FUNCTION_BLOCK FB_HeatPump EXTENDS FB_Actor2Point
VAR_INPUT
END_VAR
VAR_OUTPUT
END_VAR
VAR
	//I/O Links
	bSetStatusOn_OUT 	AT %Q* : BOOL := FALSE;
END_VAR

SelectControlMode();

METHOD SetState_BO : BOOL
VAR_INPUT
END_VAR
//output
bSetStatusOn_OUT := bSetStatusOn;
END_METHOD

END_FUNCTION_BLOCK

(* stored: Version 1.1.0.1, ProductVersion 3.1.4024.9
   POU FB_HeatPump: Id {6be2a86b-9314-45b6-a0b8-c7e56c6270da}, SpecialFunc None
   Method SetState_BO: Id {d936418b-3361-4568-804e-f0c81650d572} *)
